{attribute 'linkalways'} 
{attribute 'no_explicit_call' := 'This FB is a CLASS and must be accessed using methods or properties'}
{attribute 'enable_dynamic_creation'}
FUNCTION_BLOCK Node_F_VN_FillEllipse EXTENDS VisionNode
VAR
    stEllipse : _TcVnRotatedRectangle;
    ipDestImage : _ITcVnImage;
    aColor : _TcVnVector4_LREAL;
    hrPrev : _HRESULT(S_OK);
	hresult : _HRESULT(S_OK);
END_VAR

METHOD PUBLIC  Clone : I_Node
VAR
	pNode : POINTER TO Node_F_VN_FillEllipse;
END_VAR
pNode := __NEW(Node_F_VN_FillEllipse);
Clone := pNode^;
END_METHOD

METHOD FB_init : BOOL
VAR_INPUT
	bInitRetains : BOOL; // if TRUE, the retain variables are initialized (warm start / cold start)
	bInCopyCode : BOOL;  // if TRUE, the instance afterwards gets moved into the copy code (online change)
END_VAR
AddInput('stEllipse', stEllipse);
AddInput('ipDestImage', ipDestImage);
AddInput('aColor', aColor);
AddInput('hrPrev', hrPrev);
AddOutput('ipDestImage', ipDestImage);
AddOutput('hresult',hresult);
END_METHOD

METHOD PROTECTED  OnExecute : HRESULT
hresult.Value := F_VN_FillEllipse(
    stEllipse := stEllipse.Value,
	ipDestImage := ipDestImage.Value,
    aColor := aColor.Value,
	hrPrev:= hrPrev.Value);
END_METHOD

METHOD PUBLIC PreExecutionCheck
VAR_INPUT
	Check : I_PreExecutionChecks;
END_VAR
Check.IsTrue(ipDestImage.IsValid, 'ipDestImage must contain an image');
END_METHOD

END_FUNCTION_BLOCK

(* stored: Version 1.1.0.1, ProductVersion 3.1.4024.13
   POU Node_F_VN_FillEllipse: Id {a90c6302-3ef6-06a1-17e0-338a57fb1c2d}, SpecialFunc None
   Folder Constructor: Id {37d407ac-b0e6-0f97-0647-db9b88603bb3}
   Method Clone: Id {ee31518e-afe2-0395-3c5a-d1eb58d81d56}
   Method FB_init: Id {883f7151-1939-0b23-0bf5-cfe03b479140}
   Method OnExecute: Id {964eb2a7-ce04-0baf-389a-2f65460787f0}
   Method PreExecutionCheck: Id {51fbb59f-3461-0a3a-1c6a-3ffc78afa554} *)
